SUBAPPLICATION Uebung_010b1 (* AuxFunction2_X1 auf DigitalOutput_Q1 *)
  (* Standard: 61499-2 *)
  (* Version 1.0, 2023-10-23, franz *)
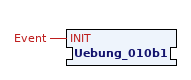
  EVENT_INPUT
    INIT;
  END_EVENT
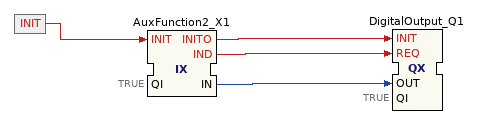
  FBS
    DigitalOutput_Q1 : QX(QI := TRUE);
    AuxFunction2_X1 : IX(QI := TRUE);
  END_FBS
  EVENT_CONNECTIONS
    INIT TO AuxFunction2_X1.INIT;
    AuxFunction2_X1.INITO TO DigitalOutput_Q1.INIT;
    AuxFunction2_X1.IND TO DigitalOutput_Q1.REQ;
  END_CONNECTIONS
  DATA_CONNECTIONS
    AuxFunction2_X1.IN TO DigitalOutput_Q1.OUT;
  END_CONNECTIONS
END_SUBAPPLICATION
